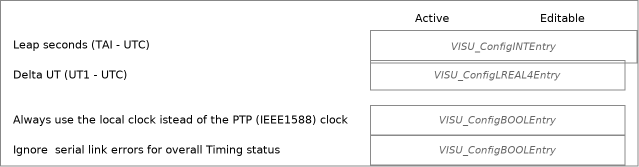
VISUALIZATION VISU_ServicesConfig_Timing  // 639x167
VAR_IN_OUT
    editableConfig : ServicesTimingConfig;
	activeConfig : ServicesTimingConfig;
END_VAR
    Frame (370,30 267x33)
        shows VISU_ConfigINTEntry(active := activeConfig.leapSeconds, editable := editableConfig.leapSeconds)
    Label (10,30 195x30), "Leap seconds (TAI - UTC)"
    Frame (370,105 255x30)
        shows VISU_ConfigBOOLEntry(active := activeConfig.alwaysUseLocalClock, editable := editableConfig.alwaysUseLocalClock)
    Label (370,5 125x27), "Active"
    Label (500,5 125x27), "Editable"
    Label (10,105 360x30), "Always use the local clock istead of the PTP (IEEE1588) clock"
    Frame (370,135 255x30)
        shows VISU_ConfigBOOLEntry(active := activeConfig.ignoreSerialError, editable := editableConfig.ignoreSerialError)
    Label (10,135 365x30), "Ignore serial link errors for overall Timing status"
    Frame (370,60 255x30)
        shows VISU_ConfigLREAL4Entry(active := activeConfig.dut, editable := editableConfig.dut)
    Label (10,60 195x30), "Delta UT (UT1 - UTC)"
END_VISUALIZATION

(* stored: Version 1.1.0.1, ProductVersion 3.1.4019.2
   Visu VISU_ServicesConfig_Timing: Id {cde25e8b-54cc-4528-bc85-d58ba5ce3967} *)
